// TIA Portal V17 export
// export: Created 2023-12-22T15:28:36.7831186Z, ExportSetting WithDefaults, DisplayName Totally Integrated Automation Portal, DisplayVersion V17, DisplayName TIA Portal Openness, DisplayVersion V17, DisplayName TIA Portal Version Control Interface, DisplayVersion V17, DisplayName STEP 7 Professional, DisplayVersion V17, DisplayName STEP 7 Safety, DisplayVersion V17, DisplayName WinCC Advanced, DisplayVersion V17
DATA_BLOCK "DOx_1_DB"   // DB210
VERSION : 0.1
// stored: AutoNumber false, DBAccessibleFromOPCUA true, InstanceOfName DOx_1, InstanceOfType FB
"DOx_1"
   // VAR RETAIN
   //    command_1 { S7_SetPoint := 'True'} : "DO_ex";
   //    command_2 { S7_SetPoint := 'True'} : "DO_ex";
   //    command_3 { S7_SetPoint := 'True'} : "DO_ex";
   //    command_4 { S7_SetPoint := 'True'} : "DO_ex";
   //    command_5 { S7_SetPoint := 'True'} : "DO_ex";
   //    command_6 { S7_SetPoint := 'True'} : "DO_ex";
   //    command_7 { S7_SetPoint := 'True'} : "DO_ex";
   //    command_8 { S7_SetPoint := 'True'} : "DO_ex";
   //    command_9 { S7_SetPoint := 'True'} : "DO_ex";
   //    command_10 { S7_SetPoint := 'True'} : "DO_ex";
   //    command_11 { S7_SetPoint := 'True'} : "DO_ex";
   //    command_12 { S7_SetPoint := 'True'} : "DO_ex";
   //    Time_DTL { S7_SetPoint := 'True'} : DTL;
   // END_VAR
BEGIN
END_DATA_BLOCK
